// TIA Portal V16 export
// export: Created 2023-03-29T11:03:46.500033Z, ExportSetting WithDefaults, DisplayName Totally Integrated Automation Portal, DisplayVersion V16 Update 6, DisplayName TIA Portal Version Control Interface, DisplayVersion V16 Update 2, DisplayName TIA Portal Openness, DisplayVersion V16 Update 6, DisplayName STEP 7 Professional, DisplayVersion V16 Update 6, DisplayName STEP 7 Safety, DisplayVersion V16, DisplayName WinCC Advanced, DisplayVersion V16 Update 6
VAR_GLOBAL   // PLC tag table "Alarm_error"
   errorAnlog_Z10 AT %M9.3 : Bool;   // sygnał błędu sygnału analogowego położenia Z10
   outAlarm AT %M1030.3 : Bool;   // Znacznik alarmu zbiorczego (Sygnalizator)
   float_min_tank_4 AT %M47.4 : Bool;   // pływak min zbiornik 4
   float_min_tank_1 AT %M47.1 : Bool;   // pływak min zbiornik 1
   float_min_tank_3 AT %M47.3 : Bool;   // pływak min zbiornik 3
   float_min_tank_2 AT %M47.2 : Bool;   // pływak min zbiornik 2
   "I2.7" AT %I2.7 : Bool;
   "I3.0" AT %I3.0 : Bool;
   "I2.6" AT %I2.6 : Bool;
   "I2.5" AT %I2.5 : Bool;
   Communication_alarm_tcp AT %M1030.2 : Bool;   // Znacznik błedu komunikacji HMI - PLC
   comunication_alarm_modbus_rtu AT %M1030.4 : Bool;   // kontrola przebiegu pętli odczytu parametró z modbus rtu
   Led_Error AT %M91.0 : Bool;   // bit sygnalizacji zapalenia led error na CPU
   Status_QRY AT %MW302 : Word;   // Status słowa przerwań (bit 0 - informacja o CPU 0- RUN, 1- Rozruch)
   statusCPU AT %M302.0 : Bool;   // 0- Run 1-Rozruch
   Error_QRY AT %MW300 : Int;   // Słowo błędu przetwarzania przerwań czasowych
   setAlarmNiskie_magistrala AT %M91.2 : Bool;   // bit alarmu niskiego ciśnienia na magistrali
   resetAlarmNiskie_magistrala AT %M91.3 : Bool;   // bit końca niskiego ciśnienia magistrala
   float_max_tank_3 AT %M46.6 : Bool;   // pływak max zbiornik 3
   float_max_tank_1 AT %M46.4 : Bool;   // pływak max zbiornik 1
   setControl_alarm_B5 AT %M91.4 : Bool;   // Załczenie sterowania zbiornikami w trybie awarii na magistrali
   float_max_tank_2 AT %M46.5 : Bool;   // pływak max zbiornik 2
   float_max_tank_4 AT %M46.7 : Bool;   // pływak max zbiornik 2
   reset_error_hwork AT %M45.6 : Bool;   // reset po błędzie gdy wszystkie zbiorniki ten sam czas pracy
END_VAR
